Fanuc KAREL source: NM0167.KL

-- PROVISIONAL review KL for V770-1; original PC SHA256 436a3277d312498a4ad3e75581d4f32a97ab3e7cb59bc810a21c0581b1db9dc3
-- Incomplete behavior may be omitted. Consult companion uncertainty JSON. Do not deploy.
PROGRAM NM0167
%NOLOCKGROUP
-- UNRESOLVED_LOCAL_POOL 5 cells at code offset 71; source declarations unknown
-- DIRECT_LOCAL_WORD_ACCESS alone does not prove INTEGER, REAL, or BOOLEAN
BEGIN
  -- UNRESOLVED_PC offsets 0-1; opcodes 7B
  -- UNRESOLVED_PC offsets 6-18; opcodes 2D,9D,52,7F
  -- UNRESOLVED_PC offsets 23-28; opcodes 7F,7B
  -- UNRESOLVED_PC offsets 33-49; opcodes 2D,2E,69,7F
  -- UNRESOLVED_PC offsets 54-76; opcodes 7F,2B,2C,7B
  -- UNRESOLVED_PC offsets 81-88; opcodes 9D,23
  -- UNRESOLVED_PC offsets 93-104; opcodes 2E,23
  -- UNRESOLVED_PC offsets 109-120; opcodes 2E,23
  -- UNRESOLVED_PC offsets 125-136; opcodes 2E,23
  -- UNRESOLVED_PC offsets 141-148; opcodes 9D,23
  -- UNRESOLVED_PC offsets 153-162; opcodes 3F,75
  -- UNRESOLVED_PC offsets 167-181; opcodes 2E,22,9D,33,35
  -- UNRESOLVED_PC offsets 186-200; opcodes 2E,22,9D,33,35
  -- UNRESOLVED_PC offsets 205-226; opcodes 27,27,27,22,AA,64,76,23
  -- UNRESOLVED_PC offsets 231-235; opcodes 7F
  -- UNRESOLVED_PC offsets 240-244; opcodes 27,AA
  -- UNRESOLVED_PC offsets 249-253; opcodes 7F
END NM0167
